FUNCTION_BLOCK SYMLINKMULTIVARSRC_277E97BEC1451D2C (* Multiple variables single value symbolic link source FB *)
  (* Standard: 61499-2 *)
  (* Version 1.0, 2008-10-02, milos, nxtControl GmbH, template *)
  PACKAGE UAO.Hackathon;
  (* Compiler Cpp *)
  {SET_ATTRIBUTE(Runtime.FBType.ImplementingType, Runtime.System#DYNGEN_SYMLINKMVAR)}
  {SET_ATTRIBUTE(Configuration.GenericFBType.InterfaceParams, Runtime.System#I:=2;VALUE${I$}:BOOL,BOOL)}
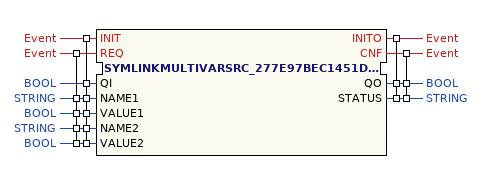
  EVENT_INPUT
    INIT WITH QI, NAME1, NAME2, VALUE1, VALUE2; (* Initializes the symbolic link data source FB with N (1 <= N <= 16) variables *)
    REQ WITH NAME1, NAME2, VALUE1, VALUE2; (* Data write request *)
  END_EVENT
  EVENT_OUTPUT
    INITO WITH QO, STATUS; (* Initialization confirm *)
    CNF WITH QO, STATUS; (* Confirmation of data write request *)
  END_EVENT
  VAR_INPUT
    QI : BOOL; (* INIT event input qualifier *)
    NAME1 : STRING := '$${PATH}'; (* Names a symbolic link variable *)
    VALUE1 : BOOL; (* New value(i) for the named variable element *)
    NAME2 : STRING := '$${PATH}'; (* Names a symbolic link variable *)
    VALUE2 : BOOL; (* New value(i) for the named variable element *)
  END_VAR
  VAR_OUTPUT
    QO : BOOL; (* Output event qualifier *)
    STATUS : STRING; (* FB status indicator *)
  END_VAR
  EC_STATES
    START;
  END_STATES
END_FUNCTION_BLOCK
